// TIA Portal V17 export
// export: Created 2025-06-26T06:49:33.7051743Z, ExportSetting WithDefaults, DisplayName Totally Integrated Automation Portal, DisplayVersion V17 Update 8, DisplayName TIA Portal Openness, DisplayVersion V17 Update 8, DisplayName TIA Portal Version Control Interface, DisplayVersion V17, DisplayName STEP 7 Professional, DisplayVersion V17 Update 8, DisplayName STEP 7 Safety, DisplayVersion V17 Update 6, DisplayName WinCC Advanced, DisplayVersion V17 Update 8
VAR_GLOBAL   // PLC tag table "Standard-Variable-Table"
   Clock_Byte AT %MB0 : Byte;   //    {ExternalAccessible false, ExternalVisible false, ExternalWritable false}
   Clock_10Hz AT %M0.0 : Bool;   //    {ExternalAccessible false, ExternalVisible false, ExternalWritable false}
   Clock_5Hz AT %M0.1 : Bool;   //    {ExternalAccessible false, ExternalVisible false, ExternalWritable false}
   "Clock_2.5Hz" AT %M0.2 : Bool;   //    {ExternalAccessible false, ExternalVisible false, ExternalWritable false}
   Clock_2Hz AT %M0.3 : Bool;   //    {ExternalAccessible false, ExternalVisible false, ExternalWritable false}
   "Clock_1.25Hz" AT %M0.4 : Bool;   //    {ExternalAccessible false, ExternalVisible false, ExternalWritable false}
   Clock_1Hz AT %M0.5 : Bool;   //    {ExternalAccessible false, ExternalVisible false, ExternalWritable false}
   "Clock_0.625Hz" AT %M0.6 : Bool;   //    {ExternalAccessible false, ExternalVisible false, ExternalWritable false}
   "Clock_0.5Hz" AT %M0.7 : Bool;   //    {ExternalAccessible false, ExternalVisible false, ExternalWritable false}
   System_Byte AT %MB1 : Byte;   //    {ExternalAccessible false, ExternalVisible false, ExternalWritable false}
   FirstScan AT %M1.0 : Bool;   //    {ExternalAccessible false, ExternalVisible false, ExternalWritable false}
   DiagStatusUpdate AT %M1.1 : Bool;   //    {ExternalAccessible false, ExternalVisible false, ExternalWritable false}
   AlwaysTRUE AT %M1.2 : Bool;   //    {ExternalAccessible false, ExternalVisible false, ExternalWritable false}
   AlwaysFALSE AT %M1.3 : Bool;   //    {ExternalAccessible false, ExternalVisible false, ExternalWritable false}
   CVM1 AT %IW472 : Word;   //    {ExternalAccessible false, ExternalVisible false, ExternalWritable false}
   CVM2 AT %IW474 : Word;   //    {ExternalAccessible false, ExternalVisible false, ExternalWritable false}
   ModbusOK AT %I476.0 : Bool;   //    {ExternalAccessible false, ExternalVisible false, ExternalWritable false}
END_VAR
VAR_GLOBAL CONSTANT   // user constants
   Keiner : Pip := 65535;
   "Automatische Aktualisierung" : Pip := 0;
   "TPA 1" : Pip := 1;
   "TPA 2" : Pip := 2;
   "TPA 3" : Pip := 3;
   "TPA 4" : Pip := 4;
   "TPA OB Servo" : Pip := 32768;
   "Local~MC(1)" : Hw_SubModule := 51;
   "Local~Exec(1)" : Hw_SubModule := 52;
   "Local(1)" : Hw_SubModule := 49;
   "Local~HSC_1" : Hw_Hsc := 257;
   "Local~HSC_2" : Hw_Hsc := 258;
   "Local~HSC_3" : Hw_Hsc := 259;
   "Local~HSC_4" : Hw_Hsc := 260;
   "Local~HSC_5" : Hw_Hsc := 261;
   "Local~HSC_6" : Hw_Hsc := 262;
   "Local~AI_2_AQ_2_1" : Hw_SubModule := 263;
   "Local~DI_14_DQ_10_1" : Hw_SubModule := 264;
   "Local~Pulse_1" : Hw_Pwm := 265;
   "Local~Pulse_2" : Hw_Pwm := 266;
   "Local~Pulse_3" : Hw_Pwm := 267;
   "Local~Pulse_4" : Hw_Pwm := 268;
   Engine1InPosition : Event_HwInt := 16#C0000101;
   HallSensorFlag4 : Event_HwInt := 16#C0050108;
   HallSensorFlag1 : Event_HwInt := 16#C0020108;
   HallSensorFlag2 : Event_HwInt := 16#C0030108;
   HallSensorFlag3 : Event_HwInt := 16#C0040108;
   "Sensors~KF102" : Hw_SubModule := 448;
   "Local~Common(1)" : Hw_SubModule := 50;
   "Local~Device(1)" : Hw_Device := 32;
   "Local~Configuration(1)" : Hw_SubModule := 33;
   "Local~OPC_UA" : Hw_SubModule := 117;
   "OB_Time error interrupt(1)" : OB_TIMEERROR := 80;
   "Local~DQ_8xRelay" : Hw_SubModule := 270;
   "Sensors~KF103" : Hw_SubModule := 278;
   "Sensors~KF104" : Hw_SubModule := 271;
   "Sensors~KF105" : Hw_SubModule := 272;
   "Sensors~KF106" : Hw_SubModule := 274;
   "Sensors~KF107" : Hw_SubModule := 276;
   "Sensors~KF108" : Hw_SubModule := 277;
   "Sensors~KF109" : Hw_SubModule := 279;
   "Sensors~KF110" : Hw_SubModule := 280;
   "Sensors~KF219" : Hw_SubModule := 284;
   "Sensors~KF220" : Hw_SubModule := 285;
   "Sensors~KF221" : Hw_SubModule := 286;
   "Sensors~KF222" : Hw_SubModule := 287;
   "Sensors~KF223" : Hw_SubModule := 288;
   "Sensors~KF224" : Hw_SubModule := 289;
   "Sensors~KF227" : Hw_SubModule := 292;
   "Sensors~KF225" : Hw_SubModule := 293;
   "Sensors~KF226" : Hw_SubModule := 290;
   "Sensors~KF228" : Hw_SubModule := 291;
   "Local~AI_1xRTD_1" : Hw_SubModule := 294;
   "Local~PROFINET_interface_1(1)" : Hw_Interface := 64;
   "Local~PROFINET_interface_1~Port_2(1)" : Hw_Interface := 66;
   "Local~PROFINET_interface_1~Port_1(1)" : Hw_Interface := 65;
   "Local~PROFINET_IO-System" : Hw_IoSystem := 269;
   "Sensors~Proxy" : Hw_SubModule := 441;
   "Sensors~IODevice" : Hw_Device := 275;
   "Sensors~Head" : Hw_SubModule := 442;
   "Sensors~PROFINET_interface" : Hw_Interface := 443;
   "Sensors~PROFINET_interface~Port_1" : Hw_Interface := 444;
   "Sensors~PROFINET_interface~Port_2" : Hw_Interface := 445;
   "Sensors~ET-Con_2" : Hw_SubModule := 449;
   "Sensors~ET-Con_1" : Hw_SubModule := 447;
   "Sensors~KF111" : Hw_SubModule := 281;
   "OB_Main(1)" : OB_PCYCLE := 1;
   "HBL-SC-02~Proxy" : Hw_SubModule := 283;
   "HBL-SC-02~IODevice" : Hw_Device := 273;
   "HBL-SC-02~Interface" : Hw_Interface := 295;
   "HBL-SC-02~Interface~Port_1" : Hw_Interface := 296;
   "HBL-SC-02~Interface~Port_2" : Hw_Interface := 297;
   "HBL-SC-02~Head" : Hw_SubModule := 298;
   "HBL-SC-02~PPO_Type_6_1" : Hw_SubModule := 299;
   "HBL-SC-10~Proxy" : Hw_SubModule := 302;
   "HBL-SC-10~IODevice" : Hw_Device := 300;
   "HBL-SC-10~Interface" : Hw_Interface := 303;
   "HBL-SC-10~Interface~Port_1" : Hw_Interface := 304;
   "HBL-SC-10~Interface~Port_2" : Hw_Interface := 305;
   "HBL-SC-10~Head" : Hw_SubModule := 306;
   "HBL-SC-10~PPO_Type_6_1" : Hw_SubModule := 307;
   "HBL-SC-01~Proxy" : Hw_SubModule := 310;
   "HBL-SC-01~IODevice" : Hw_Device := 308;
   "HBL-SC-01~Interface" : Hw_Interface := 311;
   "HBL-SC-01~Interface~Port_1" : Hw_Interface := 312;
   "HBL-SC-01~Interface~Port_2" : Hw_Interface := 313;
   "HBL-SC-01~Head" : Hw_SubModule := 314;
   "HBL-SC-01~PPO_Type_6_1" : Hw_SubModule := 315;
   "OB_Main_Cyclic(1)" : OB_Cyclic := 30;
END_VAR
